# EPICS SNL sequencer program: support/seq/test/validate/userfunc.st
/*************************************************************************\
Copyright (c) 2010-2015 Helmholtz-Zentrum Berlin f. Materialien
                        und Energie GmbH, Germany (HZB)
This file is distributed subject to a Software License Agreement found
in the file LICENSE that is included with this distribution.
\*************************************************************************/
program userfuncTest

%%#include "../testSupport.h"

option +s;

%{
static void incr(SS_ID ssId, int *pv, VAR_ID v);
static void incr_compat(SS_ID ssId, int *pv, VAR_ID v);
static void set_i(USER_VAR *const pVar, int value);
static void null(void);
}%

int i = 0;
assign i;

entry {
    seq_test_init(20);
}

ss myss {
    state doit {
        int i_saved = 0;
        when (delay(0.1)) {
            if (i % 2)
                incr(ssId, &i, pvIndex(i));
            else
                incr_compat(ssId, &i, pvIndex(i));
            testOk1(i_saved == i-1);
            i_saved = i;
            set_i(pVar, 1);
            testOk1(i == 1);
            null();
        } state doit
        when (i_saved == 10) {
        } exit
    }
}

exit {
    seq_test_done();
}

%{
static void incr_compat(SS_ID ssId, int *pv, VAR_ID v)
{
    seq_pvGet(ssId, v, SYNC);
    *pv += 1;
    seq_pvPut(ssId, v, SYNC);
}

static void incr(SS_ID ssId, int *pv, VAR_ID v)
{
    seq_pvGetTmo(ssId, v, SYNC, 1.0);
    *pv += 1;
    seq_pvPutTmo(ssId, v, SYNC, 1.0);
}

static void set_i(USER_VAR *const pVar, int value)
{
    pVar->i = value;
}

static void null(void)
{
}
}%
